{attribute 'linkalways'} 
{attribute 'no_explicit_call' := 'This FB is a CLASS and must be accessed using methods or properties'}
{attribute 'enable_dynamic_creation'}
FUNCTION_BLOCK FINAL ADD_LINT EXTENDS Node
VAR
	in1 : _LINT(0);
	in2 : _LINT(0);
	out : _LINT(0);
END_VAR

METHOD PUBLIC Clone : I_Node
VAR
	pNode : POINTER TO ADD_LINT;
END_VAR
pNode := __NEW(ADD_LINT);
Clone := pNode^;
END_METHOD

METHOD FB_init : BOOL
VAR_INPUT
	bInitRetains : BOOL; // if TRUE, the retain variables are initialized (warm start / cold start)
	bInCopyCode : BOOL;  // if TRUE, the instance afterwards gets moved into the copy code (online change)
END_VAR
AddInput('in1',THIS^.in1);
AddInput('in2',THIS^.in2);
AddOutput('out', THIS^.out);
END_METHOD

METHOD PROTECTED OnExecute
VAR
END_VAR
out.Value := in1.Value + in2.Value;
END_METHOD

END_FUNCTION_BLOCK

(* stored: Version 1.1.0.1, ProductVersion 3.1.4024.15
   POU ADD_LINT: Id {0126de4a-c86a-44a1-94e3-587762380c34}, SpecialFunc None
   Folder Constructor: Id {95bbfc56-bef0-490e-b068-397bb05ce4c9}
   Method Clone: Id {d7a96e97-6638-4a3f-a5ad-416eecb622dd}
   Method FB_init: Id {3190b2d8-e264-41f3-93eb-8ebebb45004c}
   Method OnExecute: Id {73f7de66-43ee-4e04-8cb5-78d38c3df2e8} *)
